(* PLC project OOP_Curso, Beckhoff Automation GmbH TwinCAT PLC Control 3.5.13.21 *)
(* stored: creationDateTime 2023-03-26T14:13:30.0192771, modificationDateTime 2023-03-26T14:13:30.0261078 *)

TYPE ST_1:
STRUCT
	sStruct : ST_2;
	sstring : STRING(80);
END_STRUCT
END_TYPE

TYPE ST_2 :
STRUCT
	bBool : BOOL;
END_STRUCT
END_TYPE

TYPE ST_Base1 :
STRUCT
	bBool1: BOOL;
	iINT : INT;
	rReal : REAL;	
END_STRUCT
END_TYPE

TYPE ST_Sub1 EXTENDS ST_Base1:
STRUCT
	ttime :TIME;
	tton  : TON;
END_STRUCT
END_TYPE

TYPE ST_Sub2 EXTENDS ST_Sub1 :
STRUCT
	bBool2: BOOL;
END_STRUCT
END_TYPE

INTERFACE I_Base1
METHOD metodo_base1 : BOOL
VAR_INPUT
END_VAR
END_METHOD
PROPERTY Prop_base1 : bool
END_PROPERTY
END_INTERFACE

INTERFACE I_Base2
METHOD metodo_base2 : BOOL
VAR_INPUT
END_VAR
END_METHOD
PROPERTY Prop_base2 : bool
END_PROPERTY
END_INTERFACE

INTERFACE I_Sub1 EXTENDS I_Base1, I_Base2
METHOD metodo_sub1 : BOOL
VAR_INPUT
END_VAR
END_METHOD
PROPERTY Prop_sub1 : BOOL
END_PROPERTY
END_INTERFACE

INTERFACE I_Sub2 EXTENDS I_Sub1
METHOD metodo_sub2 : BOOL
VAR_INPUT
END_VAR
END_METHOD
PROPERTY Prop_sub2 : BOOL
END_PROPERTY
END_INTERFACE

FUNCTION_BLOCK FB_Sub1 IMPLEMENTS I_Sub1
VAR_INPUT
END_VAR
VAR_OUTPUT
END_VAR
VAR
END_VAR

            
          

{warning 'Agregar implementación de método'}
METHOD metodo_base1 : BOOL
                  
                
END_METHOD

{warning 'Agregar implementación de método'}
METHOD metodo_base2 : BOOL
                  
                
END_METHOD

{warning 'Agregar implementación de método'}
METHOD metodo_sub1 : BOOL
                  
                
END_METHOD

{warning 'Agregar implementación de propiedad'}
PROPERTY Prop_base1 : BOOL
GET
VAR
END_VAR
                    
                  
END_GET
SET
VAR
END_VAR
                    
                  
END_SET
END_PROPERTY

{warning 'Agregar implementación de propiedad'}
PROPERTY Prop_base2 : BOOL
GET
VAR
END_VAR
                    
                  
END_GET
SET
VAR
END_VAR
                    
                  
END_SET
END_PROPERTY

{warning 'Agregar implementación de propiedad'}
PROPERTY Prop_sub1 : BOOL
GET
VAR
END_VAR
                    
                  
END_GET
SET
VAR
END_VAR
                    
                  
END_SET
END_PROPERTY
END_FUNCTION_BLOCK

FUNCTION_BLOCK FB_Sub2 IMPLEMENTS I_Sub2
VAR_INPUT
END_VAR
VAR_OUTPUT
END_VAR
VAR
END_VAR

            
          

{warning 'Agregar implementación de método'}
METHOD metodo_base1 : BOOL
                  
                
END_METHOD

{warning 'Agregar implementación de método'}
METHOD metodo_base2 : BOOL
                  
                
END_METHOD

{warning 'Agregar implementación de método'}
METHOD metodo_sub1 : BOOL
                  
                
END_METHOD

{warning 'Agregar implementación de método'}
METHOD metodo_sub2 : BOOL
                  
                
END_METHOD

{warning 'Agregar implementación de propiedad'}
PROPERTY Prop_base1 : BOOL
GET
VAR
END_VAR
                    
                  
END_GET
SET
VAR
END_VAR
                    
                  
END_SET
END_PROPERTY

{warning 'Agregar implementación de propiedad'}
PROPERTY Prop_base2 : BOOL
GET
VAR
END_VAR
                    
                  
END_GET
SET
VAR
END_VAR
                    
                  
END_SET
END_PROPERTY

{warning 'Agregar implementación de propiedad'}
PROPERTY Prop_sub1 : BOOL
GET
VAR
END_VAR
                    
                  
END_GET
SET
VAR
END_VAR
                    
                  
END_SET
END_PROPERTY

{warning 'Agregar implementación de propiedad'}
PROPERTY Prop_sub2 : BOOL
GET
VAR
END_VAR
                    
                  
END_GET
SET
VAR
END_VAR
                    
                  
END_SET
END_PROPERTY
END_FUNCTION_BLOCK

PROGRAM _08_Herencia_Estructura_y_Interface
VAR
	//Extensión de Estructura:
	stestructura1  : ST_Sub1;
	stestructura2  : ST_Sub2;
	stestructura11 : ST_1;
	
	//Extensión de Interface:
	Sub1 : FB_Sub1;
	Sub2 : FB_Sub2;
	bBool : BOOL;

END_VAR

            //Extensión de Estructura:
stestructura1.bBool1;
stestructura1.iINT;
stestructura1.rReal;
stestructura1.ttime;
stestructura1.tton(in:= TRUE, pt:=T#1S);

stestructura2.bBool1;
stestructura2.iINT;
stestructura2.rReal;
stestructura2.ttime;
stestructura2.tton(in:= TRUE, pt:=T#1S);
stestructura2.bBool2;


stestructura11.sstring;
stestructura11.sStruct.bBool;

//Extensión de Interface:
Sub1.metodo_base1();
Sub1.Prop_base1;
Sub1.Prop_base1 := bBool;

Sub2.metodo_sub2();
Sub2.Prop_base2;
Sub1.Prop_base2 := bBool;
          
END_PROGRAM
